% RSLogix 500 project P4A_WATER_TREATMENT_SYSTEM.RSS, saved by version 8.30.00.16 %
PROJECT "TREATER"    % processor: Bul.1763 MicroLogix 1100 Series B %

PROGRAM FILES
  LAD 2 "MAIN"  4 rungs
  LAD 3 "IO"  7 rungs
  LAD 4 "POSITION"  10 rungs
  LAD 5 "CONTROL"  10 rungs

DATA FILES
  O0 OUTPUT  4 elements
  I1 INPUT  6 elements
  S2 STATUS  66 elements
  B3 BINARY  2 elements
  T4 TIMER  4 elements
  C5 COUNTER  1 elements
  R6 CONTROL  1 elements
  N7 INTEGER  2 elements
  F8 FLOAT  1 elements
  MG9 MESSAGE  1 elements

LADDER 2 "MAIN"
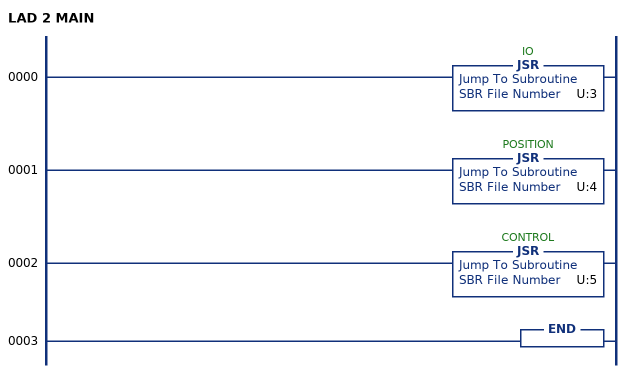
% Rung: 0 %
SOR JSR U:3 EOR
%   U:3  "IO" %
% Rung: 1 %
SOR JSR U:4 EOR
%   U:4  "POSITION" %
% Rung: 2 %
SOR JSR U:5 EOR
%   U:5  "CONTROL" %
% Rung: 3 %
SOR END EOR

LADDER 3 "IO"
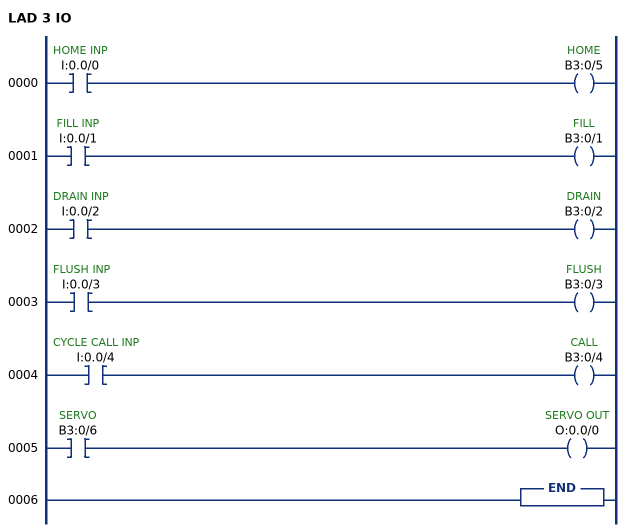
% Rung: 0 %
SOR XIC I:0.0/0 OTE B3:0/5 EOR
%   I:0.0/0  "HOME INP" %
%   B3:0/5  "HOME" %
% Rung: 1 %
SOR XIC I:0.0/1 OTE B3:0/1 EOR
%   I:0.0/1  "FILL INP" %
%   B3:0/1  "FILL" %
% Rung: 2 %
SOR XIC I:0.0/2 OTE B3:0/2 EOR
%   I:0.0/2  "DRAIN INP" %
%   B3:0/2  "DRAIN" %
% Rung: 3 %
SOR XIC I:0.0/3 OTE B3:0/3 EOR
%   I:0.0/3  "FLUSH INP" %
%   B3:0/3  "FLUSH" %
% Rung: 4 %
SOR XIC I:0.0/4 OTE B3:0/4 EOR
%   I:0.0/4  "CYCLE CALL INP" %
%   B3:0/4  "CALL" %
% Rung: 5 %
SOR XIC B3:0/6 OTE O:0.0/0 EOR
%   B3:0/6  "SERVO" %
%   O:0.0/0  "SERVO OUT" %
% Rung: 6 %
SOR END EOR

LADDER 4 "POSITION"
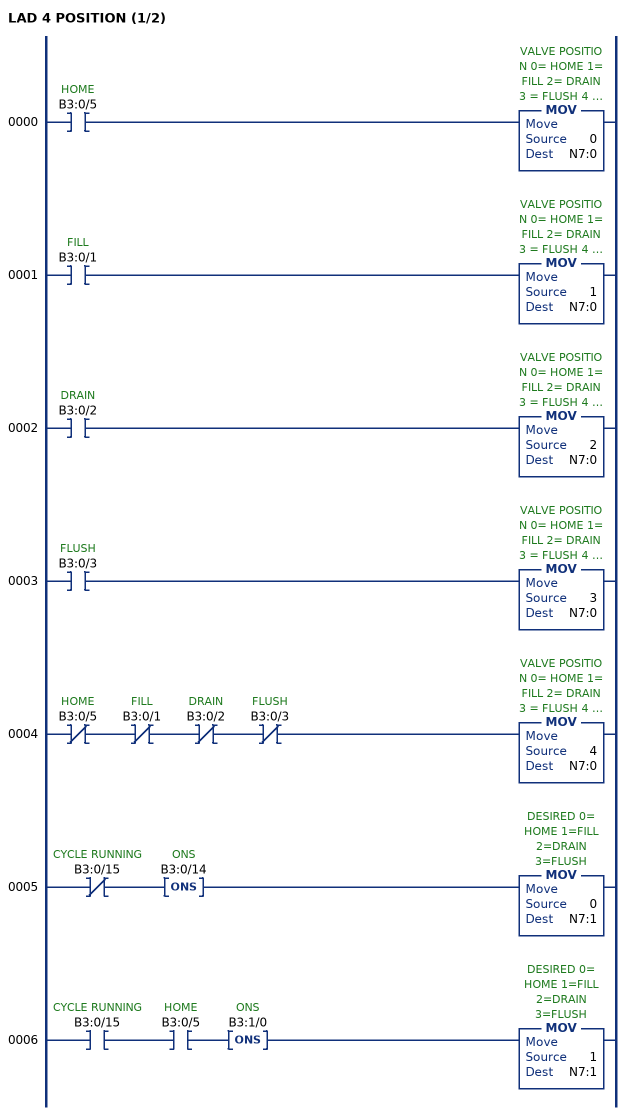
% Rung: 0 %
SOR XIC B3:0/5 MOV 0 N7:0 EOR
%   B3:0/5  "HOME" %
%   N7:0  "VALVE POSITION 0= HOME 1= FILL 2= DRAIN 3 = FLUSH 4 = TRAVELLING" %
% Rung: 1 %
SOR XIC B3:0/1 MOV 1 N7:0 EOR
%   B3:0/1  "FILL" %
%   N7:0  "VALVE POSITION 0= HOME 1= FILL 2= DRAIN 3 = FLUSH 4 = TRAVELLING" %
% Rung: 2 %
SOR XIC B3:0/2 MOV 2 N7:0 EOR
%   B3:0/2  "DRAIN" %
%   N7:0  "VALVE POSITION 0= HOME 1= FILL 2= DRAIN 3 = FLUSH 4 = TRAVELLING" %
% Rung: 3 %
SOR XIC B3:0/3 MOV 3 N7:0 EOR
%   B3:0/3  "FLUSH" %
%   N7:0  "VALVE POSITION 0= HOME 1= FILL 2= DRAIN 3 = FLUSH 4 = TRAVELLING" %
% Rung: 4 %
SOR XIO B3:0/5 XIO B3:0/1 XIO B3:0/2 XIO B3:0/3 MOV 4 N7:0 EOR
%   B3:0/5  "HOME" %
%   B3:0/1  "FILL" %
%   B3:0/2  "DRAIN" %
%   B3:0/3  "FLUSH" %
%   N7:0  "VALVE POSITION 0= HOME 1= FILL 2= DRAIN 3 = FLUSH 4 = TRAVELLING" %
% Rung: 5 %
SOR XIO B3:0/15 ONS B3:0/14 MOV 0 N7:1 EOR
%   B3:0/15  "CYCLE RUNNING" %
%   B3:0/14  "ONS" %
%   N7:1  "DESIRED 0= HOME 1=FILL 2=DRAIN 3=FLUSH" %
% Rung: 6 %
SOR XIC B3:0/15 XIC B3:0/5 ONS B3:1/0 MOV 1 N7:1 EOR
%   B3:0/15  "CYCLE RUNNING" %
%   B3:0/5  "HOME" %
%   B3:1/0  "ONS" %
%   N7:1  "DESIRED 0= HOME 1=FILL 2=DRAIN 3=FLUSH" %

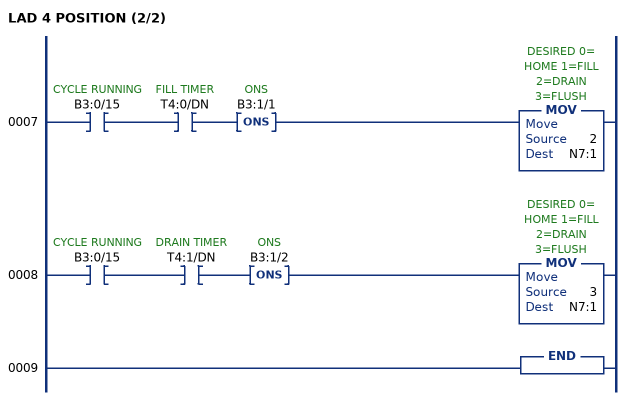
% Rung: 7 %
SOR XIC B3:0/15 XIC T4:0/DN ONS B3:1/1 MOV 2 N7:1 EOR
%   B3:0/15  "CYCLE RUNNING" %
%   T4:0  "FILL TIMER" %
%   B3:1/1  "ONS" %
%   N7:1  "DESIRED 0= HOME 1=FILL 2=DRAIN 3=FLUSH" %
% Rung: 8 %
SOR XIC B3:0/15 XIC T4:1/DN ONS B3:1/2 MOV 3 N7:1 EOR
%   B3:0/15  "CYCLE RUNNING" %
%   T4:1  "DRAIN TIMER" %
%   B3:1/2  "ONS" %
%   N7:1  "DESIRED 0= HOME 1=FILL 2=DRAIN 3=FLUSH" %
% Rung: 9 %
SOR END EOR

LADDER 5 "CONTROL"
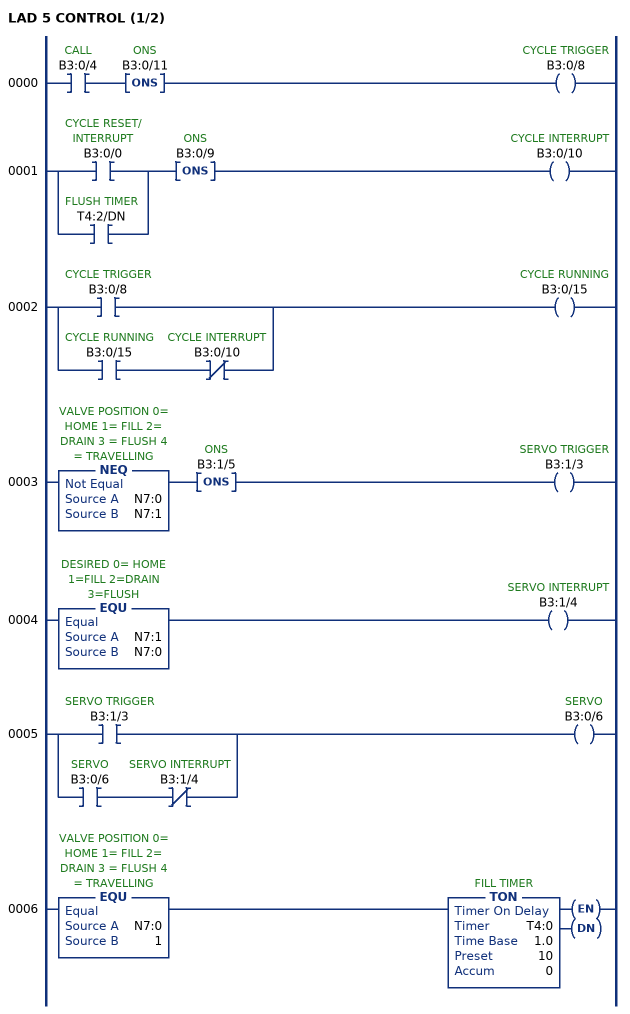
% Rung: 0 %
SOR XIC B3:0/4 ONS B3:0/11 OTE B3:0/8 EOR
%   B3:0/4  "CALL" %
%   B3:0/11  "ONS" %
%   B3:0/8  "CYCLE TRIGGER" %
% Rung: 1 %
SOR BST XIC B3:0/0 NXB XIC T4:2/DN BND ONS B3:0/9 OTE B3:0/10 EOR
%   B3:0/0  "CYCLE RESET/INTERRUPT" %
%   T4:2  "FLUSH TIMER" %
%   B3:0/9  "ONS" %
%   B3:0/10  "CYCLE INTERRUPT" %
% Rung: 2 %
SOR BST XIC B3:0/8 NXB XIC B3:0/15 XIO B3:0/10 BND OTE B3:0/15 EOR
%   B3:0/8  "CYCLE TRIGGER" %
%   B3:0/15  "CYCLE RUNNING" %
%   B3:0/10  "CYCLE INTERRUPT" %
% Rung: 3 %
SOR NEQ N7:0 N7:1 ONS B3:1/5 OTE B3:1/3 EOR
%   N7:0  "VALVE POSITION 0= HOME 1= FILL 2= DRAIN 3 = FLUSH 4 = TRAVELLING" %
%   N7:1  "DESIRED 0= HOME 1=FILL 2=DRAIN 3=FLUSH" %
%   B3:1/5  "ONS" %
%   B3:1/3  "SERVO TRIGGER" %
% Rung: 4 %
SOR EQU N7:1 N7:0 OTE B3:1/4 EOR
%   N7:1  "DESIRED 0= HOME 1=FILL 2=DRAIN 3=FLUSH" %
%   N7:0  "VALVE POSITION 0= HOME 1= FILL 2= DRAIN 3 = FLUSH 4 = TRAVELLING" %
%   B3:1/4  "SERVO INTERRUPT" %
% Rung: 5 %
SOR BST XIC B3:1/3 NXB XIC B3:0/6 XIO B3:1/4 BND OTE B3:0/6 EOR
%   B3:1/3  "SERVO TRIGGER" %
%   B3:0/6  "SERVO" %
%   B3:1/4  "SERVO INTERRUPT" %
% Rung: 6 %
SOR EQU N7:0 1 TON T4:0 1.0 10 0 EOR
%   N7:0  "VALVE POSITION 0= HOME 1= FILL 2= DRAIN 3 = FLUSH 4 = TRAVELLING" %
%   T4:0  "FILL TIMER" %

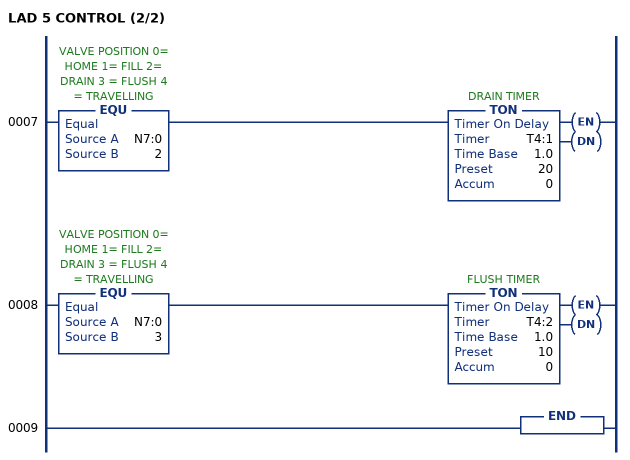
% Rung: 7 %
SOR EQU N7:0 2 TON T4:1 1.0 20 0 EOR
%   N7:0  "VALVE POSITION 0= HOME 1= FILL 2= DRAIN 3 = FLUSH 4 = TRAVELLING" %
%   T4:1  "DRAIN TIMER" %
% Rung: 8 %
SOR EQU N7:0 3 TON T4:2 1.0 10 0 EOR
%   N7:0  "VALVE POSITION 0= HOME 1= FILL 2= DRAIN 3 = FLUSH 4 = TRAVELLING" %
%   T4:2  "FLUSH TIMER" %
% Rung: 9 %
SOR END EOR

OTHER DOCUMENTED ADDRESSES
  B3:0/13  "CYCLE RESET"
  F  "FF F F F FF"
  FF  "F F F FF F"
  U2  

DATA TABLE (non-zero values as saved)
DATA B3
% B3:0 % 0X5020 0X0010
DATA T4
% .PRE .ACC %
% T4:0 % 10 0
% T4:1 % 20 0
% T4:2 % 10 0
